// Digital output FB
FUNCTION_BLOCK FB_DigitalOut EXTENDS FB_DIO IMPLEMENTS I_DigitalOut
VAR
	ibDirectControl	AT %I*	: BOOL;								// Linked input variable
	obOut			AT %Q*	: BOOL;								// Linked output variable
	eCommand				: E_DOCommand := E_DOCommand.None;	// Command received by digital output
	eState					: E_DOState	:= E_DOState.Idle;		// State of the digital output
	tBlinkPeriod			: TIME := T#2S;						// Square wave period when blinking
	tFlashTime				: TIME := T#2S;						// Time to toggle output when flashing
END_VAR
VAR RETAIN
	nSwitchCount			: UDINT;							// Counter for the number of times the input has switched (0-4294967295)
END_VAR

// Returns the blinking period
PROPERTY BlinkPeriod : TIME
GET
BlinkPeriod := tBlinkPeriod;
END_GET
END_PROPERTY

// Get the command issued to the digital output
PROPERTY Command : E_DOCommand
GET
Command := eCommand;
END_GET
END_PROPERTY

// Set the direct control value
PROPERTY DirectControl : BOOL
SET
ibDirectControl := DirectControl;
END_SET
END_PROPERTY

// Run this method every cycle
METHOD Execute
VAR_INST
	bDirectControlPrevious	: BOOL;					// Previous direct control value
	eFlashStep				: E_DOFlashStep;		// Step when flashing
	fbSquareWave			: FB_SquareWave;		// Square wave generator FB
	fbFlashTimer			: TON;					// Flash timer FB
	bOutPrevious			: BOOL;					// Previous output value
	bBlinking				: BOOL;					// True if blinking
END_VAR
// Execute command
CASE eCommand OF
	E_DOCommand.None:	// Do nothing
	E_DOCommand.On:		eState := E_DOState.TurnOn;
	E_DOCommand.Off:	eState := E_DOState.TurnOff;
	E_DOCommand.Toggle:	eState := E_DOState.Toggle;
	E_DOCommand.Blink:	eState := E_DOState.Blinking;
	E_DOCommand.Flash:	eState := E_DOState.Flashing;
END_CASE

// Execute state
CASE eState OF
	E_DOState.Idle:
		// Reset variable
		bBlinking := FALSE;
		
		// Follow direct control		
		IF ibDirectControl <> bDirectControlPrevious THEN
			obOut := ibDirectControl;
			
			nSwitchCount := nSwitchCount + 1;
			
			bDirectControlPrevious := ibDirectControl;
		END_IF
	
	E_DOState.TurnOn:
		// Turn output on
		IF obOut THEN
			// Already on, nothing to do
		ELSE
			obOut := TRUE;
			
			nSwitchCount := nSwitchCount + 1;
			
			fbLogger.AddDebug(TO_STRING(eCommand));
		END_IF
		
		eState := E_DOState.Idle;
		
	E_DOState.TurnOff:
		// Turn output off
		IF obOut THEN
			obOut := FALSE;
			
			nSwitchCount := nSwitchCount + 1;
			
			fbLogger.AddDebug(TO_STRING(eCommand));
		ELSE
			// Already off, nothing to do
		END_IF
		
		eState := E_DOState.Idle;
		
	E_DOState.Toggle:
		// Toggle output
		obOut := NOT obOut;
		
		nSwitchCount := nSwitchCount + 1;
		
		fbLogger.AddDebug(TO_STRING(eCommand));
		
		eState := E_DOState.Idle;
		
	E_DOState.Blinking:
		// Blink
		fbSquareWave(tPeriod := tBlinkPeriod, bSquareWave => obOut);
		
		IF obOut <> bOutPrevious THEN
			nSwitchCount := nSwitchCount + 1;
		END_IF
		
		bOutPrevious := obOut;
		
		IF eCommand <> E_DOCommand.None AND NOT bBlinking THEN
			fbLogger.AddDebug(TO_STRING(eCommand));
		END_IF
		
		bBlinking := TRUE;
		
	E_DOState.Flashing:
		// Flash once
		CASE eFlashStep OF
			E_DOFlashStep.Start:
				// Reset timer FB
				fbFlashTimer(IN := FALSE);
				
				eFlashStep := E_DOFlashStep.ToggleOutput;
				
			E_DOFlashStep.ToggleOutput:
				// Toggle output
				// Flash = turn on if already off, turn off if already on
				obOut := NOT obOut;
				
				nSwitchCount := nSwitchCount + 1;
				
				eFlashStep := E_DOFlashStep.WaitForTimer;
				
			E_DOFlashStep.WaitForTimer:
				// Wait for timer
				fbFlashTimer(IN := TRUE, PT := tFlashTime);
				
				IF fbFlashTimer.Q THEN
					eFlashStep := E_DOFlashStep.RestoreOutput;
				END_IF
				
			E_DOFlashStep.RestoreOutput:
				// Restore output
				obOut := NOT obOut;
				
				nSwitchCount := nSwitchCount + 1;
				
				eFlashStep := E_DOFlashStep.End;
				
			E_DOFlashStep.End:
				// Reset
				eState := E_DOState.Idle;
				eFlashStep := E_DOFlashStep.Start;
		END_CASE
		
		IF eCommand <> E_DOCommand.None THEN
			fbLogger.AddDebug(TO_STRING(eCommand));
		END_IF
		
END_CASE

// Reset command
eCommand := E_DOCommand.None;
END_METHOD

// Returns the flash time
PROPERTY FlashTime : TIME
GET
FlashTime := tFlashTime;
END_GET
END_PROPERTY

// Get HMI data
PROPERTY HmiData : ST_HmiDigitalOut
GET
HmiData.sName := sName;
HmiData.eState := eState;
HmiData.bValue := obOut;
END_GET
END_PROPERTY

// Set the square wave period when blinking (default 2s)
METHOD SetBlinkPeriod
VAR_INPUT
	tPeriod		: TIME;			// Blink period
END_VAR
tBlinkPeriod := tPeriod;
END_METHOD

// Set digital output command
METHOD SetCommand
VAR_INPUT
	eCommandIn		: E_DOCommand;	// Command
END_VAR
eCommand := eCommandIn;
END_METHOD

// Set the time to toggle the output when flashing (default 2s)
METHOD SetFlashTime
VAR_INPUT
	tTime		: TIME;			// Flash time
END_VAR
tFlashTime := tTime;
END_METHOD

// Get the digital output state (enum)
PROPERTY State : E_DOState
GET
State := eState;
END_GET
END_PROPERTY

// Get the digital output boolean value
PROPERTY Value : BOOL
GET
Value := obOut;
END_GET
END_PROPERTY

END_FUNCTION_BLOCK

(* stored: Version 1.1.0.1, ProductVersion 3.1.4024.12
   POU FB_DigitalOut: Id {b35e412e-e9e8-4ab6-9166-d5ebb85f5884}, SpecialFunc None
   Folder Methods: Id {fd57294d-b22b-4b48-9c70-35554cf8bddd}
   Folder Properties: Id {d843abcd-0e9e-44d2-8a40-30e1f4591b74}
   Property BlinkPeriod: Id {d30d495d-45e2-4229-a638-97ee0f670a3b}
   Get Get: Id {473ef06b-afaf-46eb-83c6-0f97258a5543}
   Property Command: Id {ad05d6f0-03fd-40cc-be94-7ba10c9b72d2}
   Get Get: Id {cb5ec0da-2500-49a3-85f2-cec48dffd54b}
   Property DirectControl: Id {9a4318fa-8a46-4b15-bf88-2397f48b231b}
   Set Set: Id {4ff3a8ac-3d99-4bd2-93c3-e586a361bc70}
   Method Execute: Id {acc0a333-4bb0-4e2d-b2d9-43ae1aeb724a}
   Property FlashTime: Id {b749b4db-b700-45aa-bb48-3a3cd436affa}
   Get Get: Id {ec801c58-aecc-470d-ae31-07982bee2e88}
   Property HmiData: Id {449edecb-a8b0-4103-9b2e-9c4885eb3ba3}
   Get Get: Id {00921dad-3c6b-43c0-8d74-4b59645454a6}
   Method SetBlinkPeriod: Id {e22ef653-e151-48f0-be86-6f845c7b9a84}
   Method SetCommand: Id {cb5c389a-0996-427d-ac00-33ffd772358b}
   Method SetFlashTime: Id {8d1e46ea-0b38-4ff9-9b69-4c4d37ad22bd}
   Property State: Id {133b50f2-b313-40dd-a893-5ecaf720f841}
   Get Get: Id {923a5a00-f017-49cd-a547-71e0903232ef}
   Property Value: Id {a76407f9-3e84-4be9-ab25-472ebdb1fbd0}
   Get Get: Id {cf7390ab-a2d9-4024-86f3-1225fe27594a} *)
